FUNCTION_BLOCK FB_NOTT_CRYO_INTERLOCKS
VAR_INPUT
END_VAR
VAR_OUTPUT
END_VAR
VAR
		stat:		T_NOTT_STAT;
END_VAR

END_FUNCTION_BLOCK

(* stored: Version 1.1.0.1, ProductVersion 3.1.4024.14
   POU FB_NOTT_CRYO_INTERLOCKS: Id {f5954335-cc13-4f49-8d9a-cbf7fe5d073b}, SpecialFunc None *)
